Staubli VAL3: start.pgx

program start()
  local bool result
  local string msg
  local num value
  local trsf TRSF
begin
  call init()
  call login(skCamera,"admin","",nHandleCount,result)
  if result
    putln("OK")
  endIf
  call readNumValue(nHandleCount,"C",3,value,result)
  putln(value)
  call readTrsf(nHandleCount,"C",3,TRSF,result)
  if !result
    call getErrorMessage(nHandleCount,msg)
    put(msg)
  endIf
  //? result
  //? TRSF
end
